SYSTEM DEV_MGT_APP (* Device Management Application Model *)
  (* Standard: 61499-1; Classification: Device Management *)
  (* Version 0.0, 2003-03-30, JHC, Rockwell Automation, Fixed missing (empty) FBD in Application. *)
  APPLICATION APP1
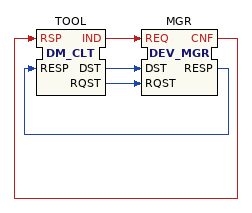
    FBS
      TOOL : DM_CLT;
      MGR : DEV_MGR;
    END_FBS
    EVENT_CONNECTIONS
      TOOL.IND TO MGR.REQ;
      MGR.CNF TO TOOL.RSP;
    END_CONNECTIONS
    DATA_CONNECTIONS
      TOOL.DST TO MGR.DST;
      TOOL.RQST TO MGR.RQST;
      MGR.RESP TO TOOL.RESP;
    END_CONNECTIONS
  END_APPLICATION
  DEVICE TOOL : FRAME_DEVICE
    RESOURCE RES1 : PANEL_RESOURCE
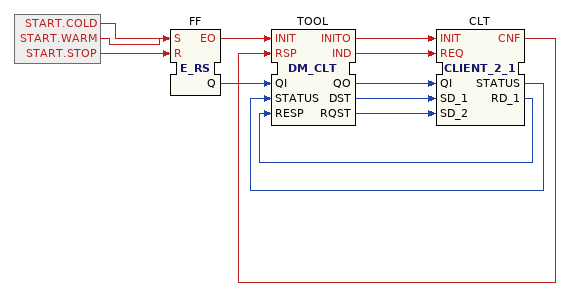
      FBS
        CLT : CLIENT_2_1;
        FF : E_RS;
        TOOL : DM_CLT;
      END_FBS
      EVENT_CONNECTIONS
        START.COLD TO FF.S;
        START.WARM TO FF.S;
        START.STOP TO FF.R;
        FF.EO TO TOOL.INIT;
        TOOL.INITO TO CLT.INIT;
        TOOL.IND TO CLT.REQ;
        CLT.CNF TO TOOL.RSP;
      END_CONNECTIONS
      DATA_CONNECTIONS
        FF.Q TO TOOL.QI;
        TOOL.QO TO CLT.QI;
        TOOL.DST TO CLT.SD_1;
        TOOL.RQST TO CLT.SD_2;
        CLT.STATUS TO TOOL.STATUS;
        CLT.RD_1 TO TOOL.RESP;
      END_CONNECTIONS
    END_RESOURCE
  END_DEVICE
  DEVICE DEV : RMT_DEV
    RESOURCE MGR : RMT_RES
    END_RESOURCE
  END_DEVICE
  MAPPINGS
    APP1.TOOL ON TOOL.RES1.TOOL;
  END_MAPPINGS
END_SYSTEM
